FUNCTION_BLOCK Safety IMPLEMENTS I_Execute
VAR_INPUT
	bFeedbackOk			: BOOL;
	bOperational		: BOOL;
END_VAR
VAR_OUTPUT
	bRun				: BOOL;
	bReset				: BOOL;
END_VAR
VAR
	_hmi				: Safety_Hmi;
	_exe				: Execute(THIS^);
	_nState				: SINT;
	_bInit				: BOOL := TRUE;
	_tonTimeout			: TON;
	SafetyStateChanged	: Signal;
END_VAR

METHOD PRIVATE _PairAllSafetyReceivers
VAR
	domIter		: DomainIter;
	iDom		: I_Domain;
	iRec		: I_Receiver;
END_VAR
WHILE IsOk(domIter.Next(iDomain => iDom)) DO
	IF IsOk(FindRec(iDom.Recs, 'OnEStop', iRec => iRec)) THEN
		SafetyStateChanged.Pair(iRec);
	END_IF
END_WHILE
END_METHOD

METHOD Execute
IF _bInit THEN
	_PairAllSafetyReceivers();
	_bInit := FALSE;
END_IF

CASE _nState OF
	0:	// INIT SAFE
		_hmi.sStatusText := 'Emergency Stop!';
		_hmi.nStatusTextColor := COL.RED.Raw;
		_hmi.bResetButtonVis := TRUE;
		SafetyStateChanged.Option('SAFE').Emit();
		_nState := 1;
		
	1:	// SAFE
		IF _hmi.bResetButton THEN
			_hmi.bResetButton := FALSE;
			IF bFeedbackOk THEN
				_nState := 2;
			END_IF
		END_IF
	2:
		_hmi.sStatusText := 'Reset in progress...';
		_hmi.bResetButtonVis := FALSE;
	
		bRun := FALSE;
		bReset := FALSE;
		_nState := 3;
	3:
		bRun := TRUE;
		_nState := 4;	
	4:
		bReset := TRUE;
		_nState := 5;
	5:
		bReset := FALSE;
		_nState := 6;
	6:	// Check if success
		_tonTimeout(IN := TRUE, PT := T#2S);
		IF _tonTimeout.Q THEN
			_tonTimeout(IN := FALSE);
			_nState := 7;
		ELSIF bOperational THEN
			_tonTimeout(IN := FALSE);
			_nState := 8;
		END_IF
	7:
		_hmi.sStatusText := 'Reset failed: System is not operational!';
		_tonTimeout(IN := TRUE, PT := T#2S);
		IF _tonTimeout.Q THEN
			_tonTimeout(IN := FALSE);
			_nState := 0;
		END_IF
		
	8:	// INIT UNSAFE
		_hmi.sStatusText := 'System Operational';
		_hmi.nStatusTextColor := COL.BLACK.Raw;
		SafetyStateChanged.Option('UNSAFE').Emit();
		_nState := 9;
	9:	// UNSAFE
		IF NOT bFeedbackOk OR NOT bOperational THEN
			_nState := 0;
		END_IF		
END_CASE
END_METHOD

METHOD ToDebug : Debug.I_Debug
ToDebug := THIS^;
END_METHOD

END_FUNCTION_BLOCK

(* stored: Version 1.1.0.1
   POU Safety: Id {b3e295d5-4f16-41d7-a844-f3b21702d931}, SpecialFunc None
   Method _PairAllSafetyReceivers: Id {4e9df51e-e3ef-4984-a35a-c8170e71f3d9}
   Method Execute: Id {0d4e5a12-faed-4f88-9050-d68ea5e4cc9f}
   Method ToDebug: Id {87a5d53b-cb96-4c5b-9462-707939772bf7} *)
